PROGRAM FUN_Write_CSV
Var
    WriteValue          : FB_Write_CSV;
END_VAR
VAR_INPUT
 InDirectory             : T_MaxString;
AX_Variables            : ARRAY [1..500] OF ST_ValuesWrite;
END_VAR


WriteValue(InDirectory := InDirectory, ParamNbColumns := 36,AX_StructureValues := AX_Variables);

END_PROGRAM

(* stored: Version 1.1.0.1, ProductVersion 3.1.4024.11
   POU FUN_Write_CSV: Id {816e0a32-1332-45e9-86c6-85f74d76957f}, SpecialFunc None *)
